{attribute 'qualified_only'}
{attribute 'strict'}
TYPE E_MachineState :
(
	IDLE := 0,
	FILLING,
	WASHING,
	DRAINING,
	COMPLETED,
	ERROR
);
END_TYPE

(* stored: Version 1.1.0.1, ProductVersion 3.1.4024.16
   DUT E_MachineState: Id {798873c1-56e0-4f77-9948-08cd1c296fe4} *)
